// Mitsubishi GX Works2 project: PLC-Servo 실습 과제 3   PLC: Q03UDV

PROGRAM MAIN
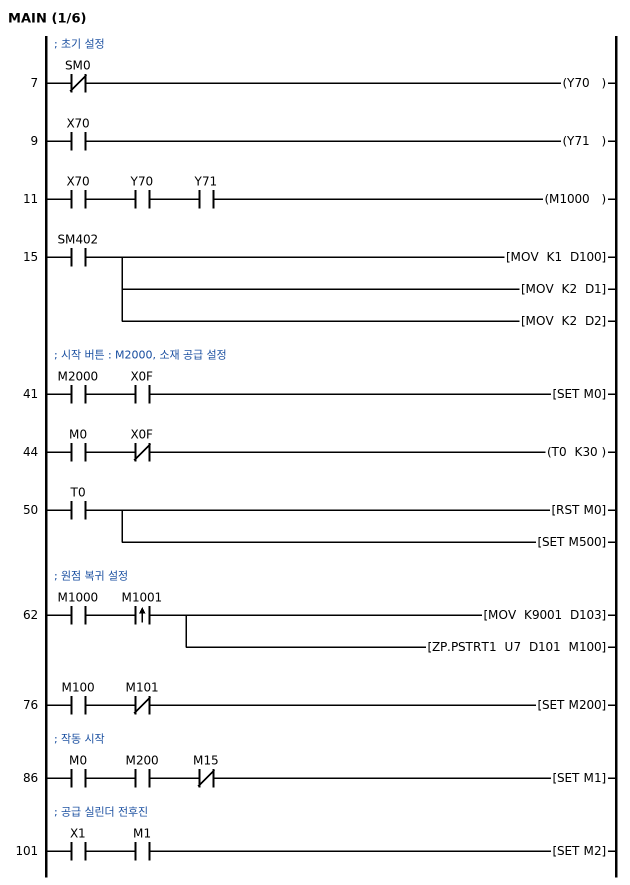
; 초기 설정
7     LDI     SM0
      OUT     Y70
9     LD      X70
      OUT     Y71
11    LD      X70
      AND     Y70
      AND     Y71
      OUT     M1000
15    LD      SM402
      MOV     K1 D100
      MOV     K2 D1
      MOV     K2 D2
; 시작 버튼 : M2000, 소재 공급 설정
41    LD      M2000
      AND     X0F
      SET     M0
44    LD      M0
      ANI     X0F
      OUT     T0 K30
50    LD      T0
      RST     M0
      SET     M500
; 원점 복귀 설정
62    LD      M1000
      ANDP    M1001
      MOV     K9001 D103
      ZP.PSTRT1 U7 D101 M100
76    LD      M100
      ANI     M101
      SET     M200
; 작동 시작
86    LD      M0
      AND     M200
      ANI     M15
      SET     M1
; 공급 실린더 전후진
101   LD      X1
      AND     M1
      SET     M2
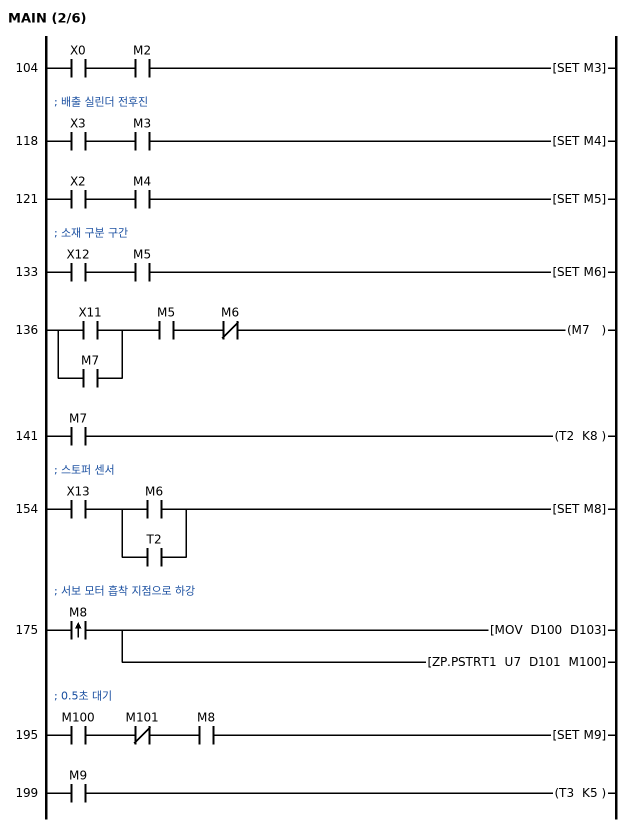
104   LD      X0
      AND     M2
      SET     M3
; 배출 실린더 전후진
118   LD      X3
      AND     M3
      SET     M4
121   LD      X2
      AND     M4
      SET     M5
; 소재 구분 구간
133   LD      X12
      AND     M5
      SET     M6
136   LD      X11
      OR      M7
      AND     M5
      ANI     M6
      OUT     M7
141   LD      M7
      OUT     T2 K8
; 스토퍼 센서
154   LD      X13
      LD      M6
      OR      T2
      ANB
      SET     M8
; 서보 모터 흡착 지점으로 하강
175   LDP     M8
      MOV     D100 D103
      ZP.PSTRT1 U7 D101 M100
; 0.5초 대기
195   LD      M100
      ANI     M101
      AND     M8
      SET     M9
199   LD      M9
      OUT     T3 K5
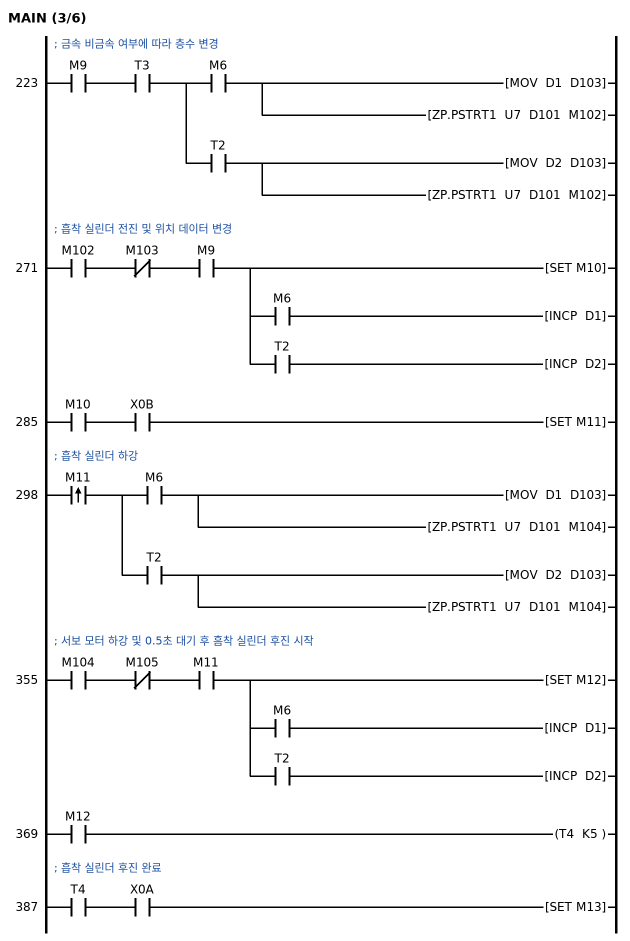
; 금속 비금속 여부에 따라 층수 변경
223   LD      M9
      AND     T3
      MPS
      AND     M6
      MOV     D1 D103
      ZP.PSTRT1 U7 D101 M102
      MPP
      AND     T2
      MOV     D2 D103
      ZP.PSTRT1 U7 D101 M102
; 흡착 실린더 전진 및 위치 데이터 변경
271   LD      M102
      ANI     M103
      AND     M9
      SET     M10
      MPS
      AND     M6
      INCP    D1
      MPP
      AND     T2
      INCP    D2
285   LD      M10
      AND     X0B
      SET     M11
; 흡착 실린더 하강
298   LDP     M11
      MPS
      AND     M6
      MOV     D1 D103
      ZP.PSTRT1 U7 D101 M104
      MPP
      AND     T2
      MOV     D2 D103
      ZP.PSTRT1 U7 D101 M104
; 서보 모터 하강 및 0.5초 대기 후 흠착 실린더 후진 시작
355   LD      M104
      ANI     M105
      AND     M11
      SET     M12
      MPS
      AND     M6
      INCP    D1
      MPP
      AND     T2
      INCP    D2
369   LD      M12
      OUT     T4 K5
; 흡착 실린더 후진 완료
387   LD      T4
      AND     X0A
      SET     M13
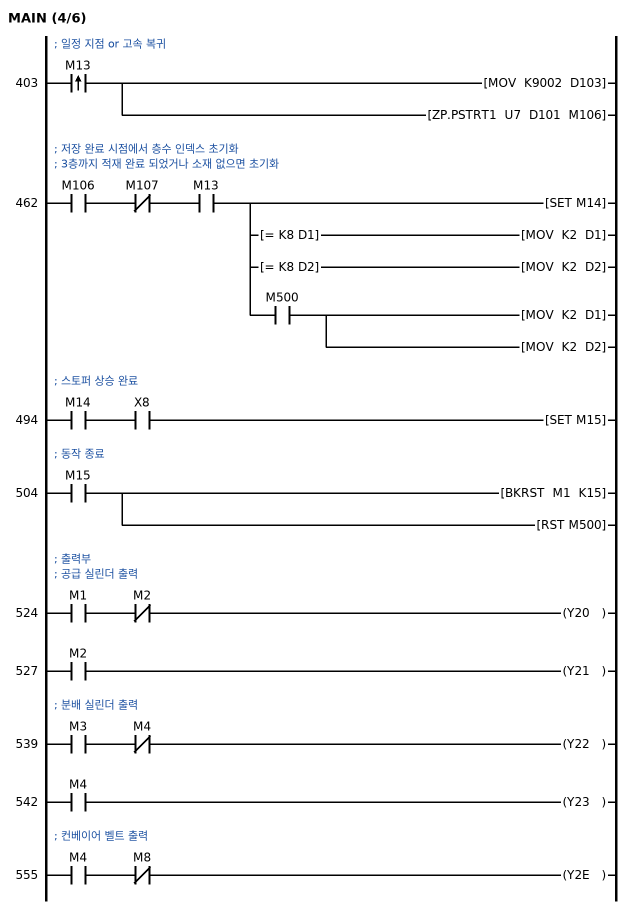
; 일정 지점 or 고속 복귀
403   LDP     M13
      MOV     K9002 D103
      ZP.PSTRT1 U7 D101 M106
; 저장 완료 시점에서 층수 인덱스 초기화
; 3층까지 적재 완료 되었거나 소재 없으면 초기화
462   LD      M106
      ANI     M107
      AND     M13
      SET     M14
      MPS
      AND=    K8 D1
      MOV     K2 D1
      MRD
      AND=    K8 D2
      MOV     K2 D2
      MPP
      AND     M500
      MOV     K2 D1
      MOV     K2 D2
; 스토퍼 상승 완료
494   LD      M14
      AND     X8
      SET     M15
; 동작 종료
504   LD      M15
      BKRST   M1 K15
      RST     M500
; 출력부
; 공급 실린더 출력
524   LD      M1
      ANI     M2
      OUT     Y20
527   LD      M2
      OUT     Y21
; 분배 실린더 출력
539   LD      M3
      ANI     M4
      OUT     Y22
542   LD      M4
      OUT     Y23
; 컨베이어 벨트 출력
555   LD      M4
      ANI     M8
      OUT     Y2E
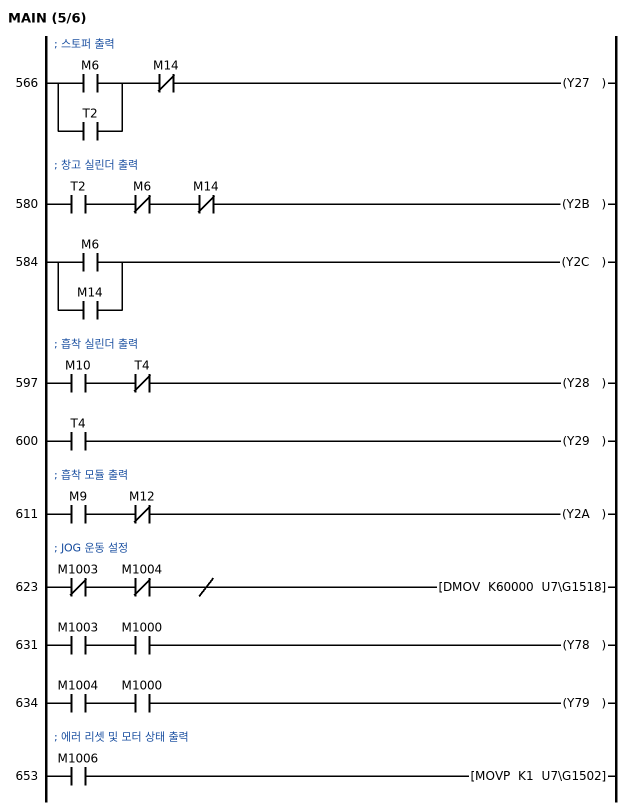
; 스토퍼 출력
566   LD      M6
      OR      T2
      ANI     M14
      OUT     Y27
; 창고 실린더 출력
580   LD      T2
      ANI     M6
      ANI     M14
      OUT     Y2B
584   LD      M6
      OR      M14
      OUT     Y2C
; 흡착 실린더 출력
597   LD      M10
      ANI     T4
      OUT     Y28
600   LD      T4
      OUT     Y29
; 흡착 모듈 출력
611   LD      M9
      ANI     M12
      OUT     Y2A
; JOG 운동 설정
623   LDI     M1003
      ANI     M1004
      INV
      DMOV    K60000 U7\G1518
631   LD      M1003
      AND     M1000
      OUT     Y78
634   LD      M1004
      AND     M1000
      OUT     Y79
; 에러 리셋 및 모터 상태 출력
653   LD      M1006
      MOVP    K1 U7\G1502
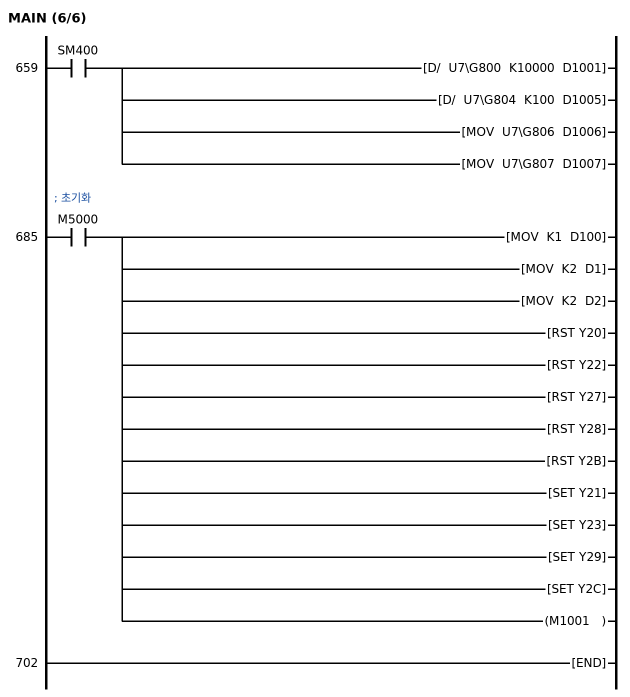
659   LD      SM400
      D/      U7\G800 K10000 D1001
      D/      U7\G804 K100 D1005
      MOV     U7\G806 D1006
      MOV     U7\G807 D1007
; 초기화
685   LD      M5000
      MOV     K1 D100
      MOV     K2 D1
      MOV     K2 D2
      RST     Y20
      RST     Y22
      RST     Y27
      RST     Y28
      RST     Y2B
      SET     Y21
      SET     Y23
      SET     Y29
      SET     Y2C
      OUT     M1001
702   END
END_PROGRAM
